// TIA Portal V17 export
// export: Created 2025-03-13T10:30:06.0846457Z, ExportSetting WithDefaults, DisplayName Totally Integrated Automation Portal, DisplayVersion V17 Update 8, DisplayName TIA Portal Openness, DisplayVersion V17 Update 8, DisplayName TIA Portal Version Control Interface, DisplayVersion V17, DisplayName SINAMICS Startdrive Advanced, DisplayVersion V17 SP2, DisplayName SINAMICS Startdrive G110M, G120, G120C, G120D, G120P, G115D, DisplayVersion V17 SP2, DisplayName SINAMICS Startdrive G130, G150, S120, S150, SINAMICS MV, S210, DisplayVersion V17 SP2, DisplayName STEP 7 Professional, DisplayVersion V17 Update 8, DisplayName SINUMERIK ONE STEP 7 Toolbox, DisplayVersion V17 Update 12, DisplayName SINUMERIK 840D sl STEP 7 Toolbox, DisplayVersion V17 Update 12, DisplayName STEP 7 Safety, DisplayVersion V17 Update 6, DisplayName WinCC Advanced, DisplayVersion V17 Update 8
FUNCTION "FC1200_UNIT_01_SEQUENCES" : Void   // FC1200, LAD
{ S7_Optimized_Access := 'FALSE' }
AUTHOR : ETXETAR
VERSION : 1.0
// stored: AutoNumber false, IsIECCheckEnabled false, SetENOAutomatically false, UDAEnableTagReadback false
BEGIN

REGION Network 1: CALL FC1203 PART CYCLE UNIT 01 CLADDING
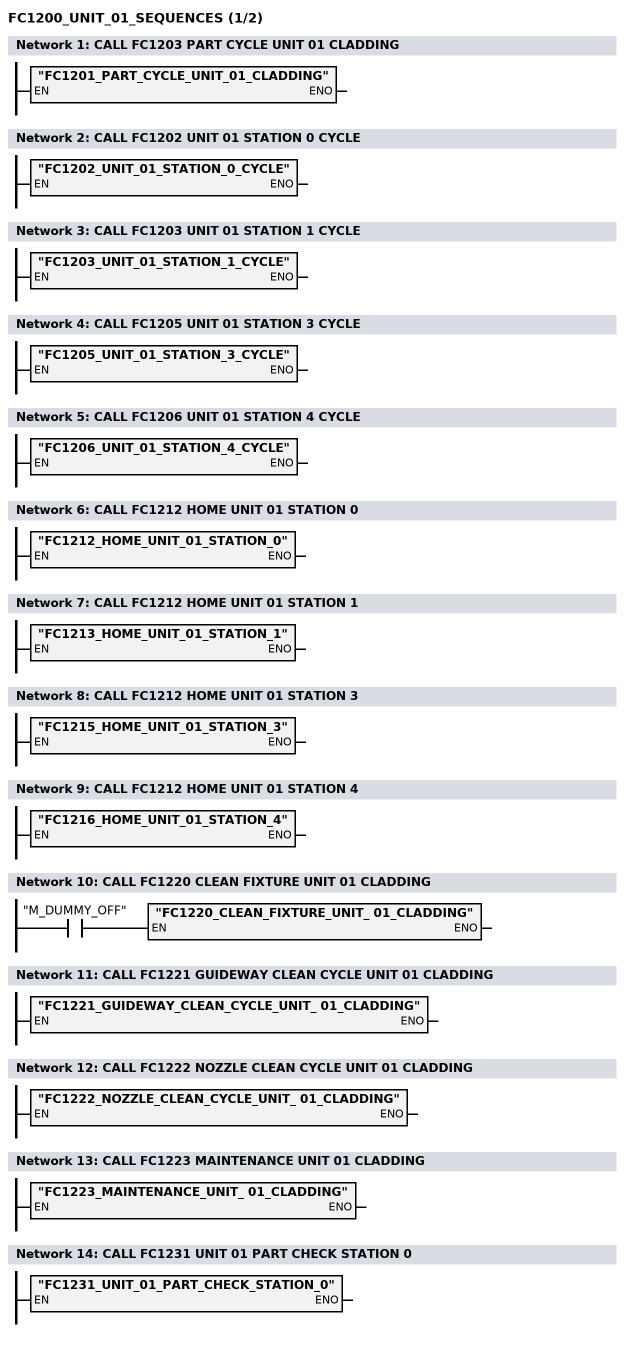
   RUNG wire#powerrail
      "FC1201_PART_CYCLE_UNIT_01_CLADDING"()
   END_RUNG
   // the same network as SCL:
   "FC1201_PART_CYCLE_UNIT_01_CLADDING"();
END_REGION

REGION Network 2: CALL FC1202 UNIT 01 STATION 0 CYCLE
   RUNG wire#powerrail
      "FC1202_UNIT_01_STATION_0_CYCLE"()
   END_RUNG
   // the same network as SCL:
   "FC1202_UNIT_01_STATION_0_CYCLE"();
END_REGION

REGION Network 3: CALL FC1203 UNIT 01 STATION 1 CYCLE
   RUNG wire#powerrail
      "FC1203_UNIT_01_STATION_1_CYCLE"()
   END_RUNG
   // the same network as SCL:
   "FC1203_UNIT_01_STATION_1_CYCLE"();
END_REGION

REGION Network 4: CALL FC1205 UNIT 01 STATION 3 CYCLE
   RUNG wire#powerrail
      "FC1205_UNIT_01_STATION_3_CYCLE"()
   END_RUNG
   // the same network as SCL:
   "FC1205_UNIT_01_STATION_3_CYCLE"();
END_REGION

REGION Network 5: CALL FC1206 UNIT 01 STATION 4 CYCLE
   RUNG wire#powerrail
      "FC1206_UNIT_01_STATION_4_CYCLE"()
   END_RUNG
   // the same network as SCL:
   "FC1206_UNIT_01_STATION_4_CYCLE"();
END_REGION

REGION Network 6: CALL FC1212 HOME UNIT 01 STATION 0
   RUNG wire#powerrail
      "FC1212_HOME_UNIT_01_STATION_0"()
   END_RUNG
   // the same network as SCL:
   "FC1212_HOME_UNIT_01_STATION_0"();
END_REGION

REGION Network 7: CALL FC1212 HOME UNIT 01 STATION 1
   RUNG wire#powerrail
      "FC1213_HOME_UNIT_01_STATION_1"()
   END_RUNG
   // the same network as SCL:
   "FC1213_HOME_UNIT_01_STATION_1"();
END_REGION

REGION Network 8: CALL FC1212 HOME UNIT 01 STATION 3
   RUNG wire#powerrail
      "FC1215_HOME_UNIT_01_STATION_3"()
   END_RUNG
   // the same network as SCL:
   "FC1215_HOME_UNIT_01_STATION_3"();
END_REGION

REGION Network 9: CALL FC1212 HOME UNIT 01 STATION 4
   RUNG wire#powerrail
      "FC1216_HOME_UNIT_01_STATION_4"()
   END_RUNG
   // the same network as SCL:
   "FC1216_HOME_UNIT_01_STATION_4"();
END_REGION

REGION Network 10: CALL FC1220 CLEAN FIXTURE UNIT 01 CLADDING
   RUNG wire#powerrail
      Contact( "M_DUMMY_OFF" )
      "FC1220_CLEAN_FIXTURE_UNIT_ 01_CLADDING"()
   END_RUNG
   // the same network as SCL:
   IF "M_DUMMY_OFF" THEN "FC1220_CLEAN_FIXTURE_UNIT_ 01_CLADDING"(); END_IF;
END_REGION

REGION Network 11: CALL FC1221 GUIDEWAY CLEAN CYCLE UNIT 01 CLADDING
   RUNG wire#powerrail
      "FC1221_GUIDEWAY_CLEAN_CYCLE_UNIT_ 01_CLADDING"()
   END_RUNG
   // the same network as SCL:
   "FC1221_GUIDEWAY_CLEAN_CYCLE_UNIT_ 01_CLADDING"();
END_REGION

REGION Network 12: CALL FC1222 NOZZLE CLEAN CYCLE UNIT 01 CLADDING
   RUNG wire#powerrail
      "FC1222_NOZZLE_CLEAN_CYCLE_UNIT_ 01_CLADDING"()
   END_RUNG
   // the same network as SCL:
   "FC1222_NOZZLE_CLEAN_CYCLE_UNIT_ 01_CLADDING"();
END_REGION

REGION Network 13: CALL FC1223 MAINTENANCE UNIT 01 CLADDING
   RUNG wire#powerrail
      "FC1223_MAINTENANCE_UNIT_ 01_CLADDING"()
   END_RUNG
   // the same network as SCL:
   "FC1223_MAINTENANCE_UNIT_ 01_CLADDING"();
END_REGION

REGION Network 14: CALL FC1231 UNIT 01 PART CHECK STATION 0
   RUNG wire#powerrail
      "FC1231_UNIT_01_PART_CHECK_STATION_0"()
   END_RUNG
   // the same network as SCL:
   "FC1231_UNIT_01_PART_CHECK_STATION_0"();
END_REGION

REGION Network 15: CALL FC1235 STATION 3 CALIBRATION UNIT 01
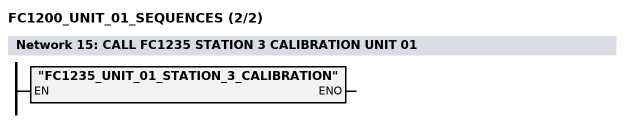
   RUNG wire#powerrail
      "FC1235_UNIT_01_STATION_3_CALIBRATION"()
   END_RUNG
   // the same network as SCL:
   "FC1235_UNIT_01_STATION_3_CALIBRATION"();
END_REGION
END_FUNCTION
